// TIA Portal V15.1 export
// export: Created 2024-05-17T05:38:39.4621169Z, ExportSetting WithDefaults, DisplayName Totally Integrated Automation Portal, DisplayVersion V15.1 Update 5, DisplayName TIA Portal Openness, DisplayVersion V15.1 Update 5, DisplayName SINAMICS Startdrive Advanced, DisplayVersion V15.1, DisplayName G130, G150, S120, S150, SINAMICS MV, S210, DisplayVersion V15.1, DisplayName G110M, G120, G120C, G120D, G120P, DisplayVersion V15.1, DisplayName STEP 7 Professional, DisplayVersion V15.1 Update 5, DisplayName STEP 7 Safety, DisplayVersion V15.1, DisplayName WinCC Professional, DisplayVersion V15.1 Update 5, DisplayName SIMATIC Visualization Architect, DisplayVersion V15.1
FUNCTION_BLOCK "LGBBodyStopper"   // FB6666, FBD
TITLE = LGBBodyStopper
{ S7_Optimized_Access := 'FALSE' }
AUTHOR : Imtech
VERSION : 0.1
// stored: AutoNumber false, IsIECCheckEnabled false, SetENOAutomatically False, UDAEnableTagReadback false
   VAR_INPUT
      I_BodyNr { ExternalAccessible := 'False'; ExternalVisible := 'False'; ExternalWritable := 'False'} : DInt;   // Body Number
      I_ColorCodeBC { ExternalAccessible := 'False'; ExternalVisible := 'False'; ExternalWritable := 'False'} : DInt;   // Color BC
      I_ColorCodeCC { ExternalAccessible := 'False'; ExternalVisible := 'False'; ExternalWritable := 'False'} : DInt;   // Color CC
      I_MMFRUSS { ExternalAccessible := 'False'; ExternalVisible := 'False'; ExternalWritable := 'False'} : DInt;   // MMFRUSS
      I_StartSearch { ExternalAccessible := 'False'; ExternalVisible := 'False'; ExternalWritable := 'False'} : Bool;   // Start search function
      I_ClearSearch { ExternalAccessible := 'False'; ExternalVisible := 'False'; ExternalWritable := 'False'} : Bool;   // Clear search result
   END_VAR
   VAR_OUTPUT
      O_BodyGo { ExternalAccessible := 'False'; ExternalVisible := 'False'; ExternalWritable := 'False'} : Bool;   // Body can GO
      O_BodyStop { ExternalAccessible := 'False'; ExternalVisible := 'False'; ExternalWritable := 'False'} : Bool;   // Body must STOP
      O_AlarmABCondition { ExternalAccessible := 'False'; ExternalVisible := 'False'; ExternalWritable := 'False'} : Bool;   // Alarm AB condition
      O_AlarmA { ExternalAccessible := 'False'; ExternalVisible := 'False'; ExternalWritable := 'False'} : Bool;   // Alarms A
      O_AlarmB { ExternalAccessible := 'False'; ExternalVisible := 'False'; ExternalWritable := 'False'} : Bool;   // Alarms B
      O_AlarmC { ExternalAccessible := 'False'; ExternalVisible := 'False'; ExternalWritable := 'False'} : Bool;   // Alarms C
      O_AlarmD { ExternalAccessible := 'False'; ExternalVisible := 'False'; ExternalWritable := 'False'} : Bool;   // Alarms D
      H_AlarmDWord { ExternalAccessible := 'False'; ExternalVisible := 'False'; ExternalWritable := 'False'} : DWord;
   END_VAR
   VAR_IN_OUT
      H_HMI : "H_HMI";   // HMI Icon Animation
      H_GBBodyStopper : "H_GBBodyStopper";   // HMI Animation
   END_VAR
   VAR DB_SPECIFIC
      AC_BodyStop { ExternalAccessible := 'False'; ExternalVisible := 'False'; ExternalWritable := 'False'} : Bool;   // Body is stopped, there is a selection active
      BodyGo { ExternalAccessible := 'False'; ExternalVisible := 'False'; ExternalWritable := 'False'} : Bool;   // Body can Go
      BodyStop { ExternalAccessible := 'False'; ExternalVisible := 'False'; ExternalWritable := 'False'} : Bool;   // Body must Stop
      HMILayerGeneral { ExternalAccessible := 'False'; ExternalVisible := 'False'; ExternalWritable := 'False'} : Bool;
      HMILayerSealing { ExternalAccessible := 'False'; ExternalVisible := 'False'; ExternalWritable := 'False'} : Bool;
      HMILayerPaint { ExternalAccessible := 'False'; ExternalVisible := 'False'; ExternalWritable := 'False'} : Bool;
      HMICmdForce { ExternalAccessible := 'False'; ExternalVisible := 'False'; ExternalWritable := 'False'} : Bool;
      HMICmdJustR { ExternalAccessible := 'False'; ExternalVisible := 'False'; ExternalWritable := 'False'} : Bool;
      HMICmdJustS2 { ExternalAccessible := 'False'; ExternalVisible := 'False'; ExternalWritable := 'False'} : Bool;
      HMICmdMM1stLayer { ExternalAccessible := 'False'; ExternalVisible := 'False'; ExternalWritable := 'False'} : Bool;
      HMICmdMM2ndLayer { ExternalAccessible := 'False'; ExternalVisible := 'False'; ExternalWritable := 'False'} : Bool;
      Status_HMICmdForce { ExternalAccessible := 'False'; ExternalVisible := 'False'; ExternalWritable := 'False'} : Bool;
      Status_HMICmdMM1stLayer { ExternalAccessible := 'False'; ExternalVisible := 'False'; ExternalWritable := 'False'} : Bool;
      Status_HMICmdMM2ndLayer { ExternalAccessible := 'False'; ExternalVisible := 'False'; ExternalWritable := 'False'} : Bool;
      Status_TABGeneral { ExternalAccessible := 'False'; ExternalVisible := 'False'; ExternalWritable := 'False'} : Bool;
      Status_TABSealing { ExternalAccessible := 'False'; ExternalVisible := 'False'; ExternalWritable := 'False'} : Bool;
      Status_TABPaint { ExternalAccessible := 'False'; ExternalVisible := 'False'; ExternalWritable := 'False'} : Bool;
      MM { ExternalAccessible := 'False'; ExternalVisible := 'False'; ExternalWritable := 'False'} : Int;
      FR { ExternalAccessible := 'False'; ExternalVisible := 'False'; ExternalWritable := 'False'} : Int;
      USS { ExternalAccessible := 'False'; ExternalVisible := 'False'; ExternalWritable := 'False'} : Int;
      FRUSS { ExternalAccessible := 'False'; ExternalVisible := 'False'; ExternalWritable := 'False'} : DInt;
      M1 { ExternalAccessible := 'False'; ExternalVisible := 'False'; ExternalWritable := 'False'} : Int;
      M2 { ExternalAccessible := 'False'; ExternalVisible := 'False'; ExternalWritable := 'False'} : Int;
      F { ExternalAccessible := 'False'; ExternalVisible := 'False'; ExternalWritable := 'False'} : Int;
      R { ExternalAccessible := 'False'; ExternalVisible := 'False'; ExternalWritable := 'False'} : Int;
      U { ExternalAccessible := 'False'; ExternalVisible := 'False'; ExternalWritable := 'False'} : Int;
      S1 { ExternalAccessible := 'False'; ExternalVisible := 'False'; ExternalWritable := 'False'} : Int;
      S2 { ExternalAccessible := 'False'; ExternalVisible := 'False'; ExternalWritable := 'False'} : Int;
      Done { ExternalAccessible := 'False'; ExternalVisible := 'False'; ExternalWritable := 'False'} : Bool;
      Error { ExternalAccessible := 'False'; ExternalVisible := 'False'; ExternalWritable := 'False'} : Bool;
      ColorCodeBCShort { ExternalAccessible := 'False'; ExternalVisible := 'False'; ExternalWritable := 'False'} : DInt;   // Color BC
      NoDuoTone { ExternalAccessible := 'False'; ExternalVisible := 'False'; ExternalWritable := 'False'} : Bool;
      DuoTone1stLayer { ExternalAccessible := 'False'; ExternalVisible := 'False'; ExternalWritable := 'False'} : Bool;
      DuoTone2ndLayer { ExternalAccessible := 'False'; ExternalVisible := 'False'; ExternalWritable := 'False'} : Bool;
      InitBit { ExternalAccessible := 'False'; ExternalVisible := 'False'; ExternalWritable := 'False'} : Bool;
      AlarmABCondition { ExternalAccessible := 'False'; ExternalVisible := 'False'; ExternalWritable := 'False'} : Bool;
      AlarmA { ExternalAccessible := 'False'; ExternalVisible := 'False'; ExternalWritable := 'False'} : Bool;
      AlarmB { ExternalAccessible := 'False'; ExternalVisible := 'False'; ExternalWritable := 'False'} : Bool;
      AlarmC { ExternalAccessible := 'False'; ExternalVisible := 'False'; ExternalWritable := 'False'} : Bool;
      AlarmD { ExternalAccessible := 'False'; ExternalVisible := 'False'; ExternalWritable := 'False'} : Bool;
      ArrayHMI_BodyNr { ExternalAccessible := 'False'; ExternalVisible := 'False'; ExternalWritable := 'False'} : Array[1..10] of DInt;
      ArrayHMI_ColorCodeBC { ExternalAccessible := 'False'; ExternalVisible := 'False'; ExternalWritable := 'False'} : Array[1..10] of Int;
      ArrayHMI_ColorCodeCC { ExternalAccessible := 'False'; ExternalVisible := 'False'; ExternalWritable := 'False'} : Array[1..10] of Int;
      ArrayHMI_MM { ExternalAccessible := 'False'; ExternalVisible := 'False'; ExternalWritable := 'False'} : Array[1..10] of Int;
      ArrayHMI_MMwithR { ExternalAccessible := 'False'; ExternalVisible := 'False'; ExternalWritable := 'False'} : Array[1..10] of Int;
      ArrayHMI_MMwithS2 { ExternalAccessible := 'False'; ExternalVisible := 'False'; ExternalWritable := 'False'} : Array[1..10] of Int;
      ArrayHMI_R { ExternalAccessible := 'False'; ExternalVisible := 'False'; ExternalWritable := 'False'} : Array[1..10] of Int;
      ArrayHMI_S2 { ExternalAccessible := 'False'; ExternalVisible := 'False'; ExternalWritable := 'False'} : Array[1..10] of Int;
      ArrayHMI_DuoTone { ExternalAccessible := 'False'; ExternalVisible := 'False'; ExternalWritable := 'False'} : Array[1..10] of Int;
      Status_BodyNr { ExternalAccessible := 'False'; ExternalVisible := 'False'; ExternalWritable := 'False'} : Array[1..10] of Bool;
      Status_ColorCodeBC { ExternalAccessible := 'False'; ExternalVisible := 'False'; ExternalWritable := 'False'} : Array[1..10] of Bool;
      Status_ColorCodeCC { ExternalAccessible := 'False'; ExternalVisible := 'False'; ExternalWritable := 'False'} : Array[1..10] of Bool;
      Status_MM { ExternalAccessible := 'False'; ExternalVisible := 'False'; ExternalWritable := 'False'} : Array[1..10] of Bool;
      Status_MMwithR { ExternalAccessible := 'False'; ExternalVisible := 'False'; ExternalWritable := 'False'} : Array[1..10] of Bool;
      Status_MMwithS2 { ExternalAccessible := 'False'; ExternalVisible := 'False'; ExternalWritable := 'False'} : Array[1..10] of Bool;
   END_VAR
   VAR
      BodyStopperSub { ExternalAccessible := 'False'; ExternalVisible := 'False'; ExternalWritable := 'False'} : "LGBBodyStopperSub";   // LBodyStopperSub
   END_VAR
   VAR_TEMP   // added for the SCL form of the ladder/FBD networks
      _w1 : Bool;
      _w2 : Bool;
   END_VAR
BEGIN

REGION Network 1: **** 1 - Inputs **** Layer INIT
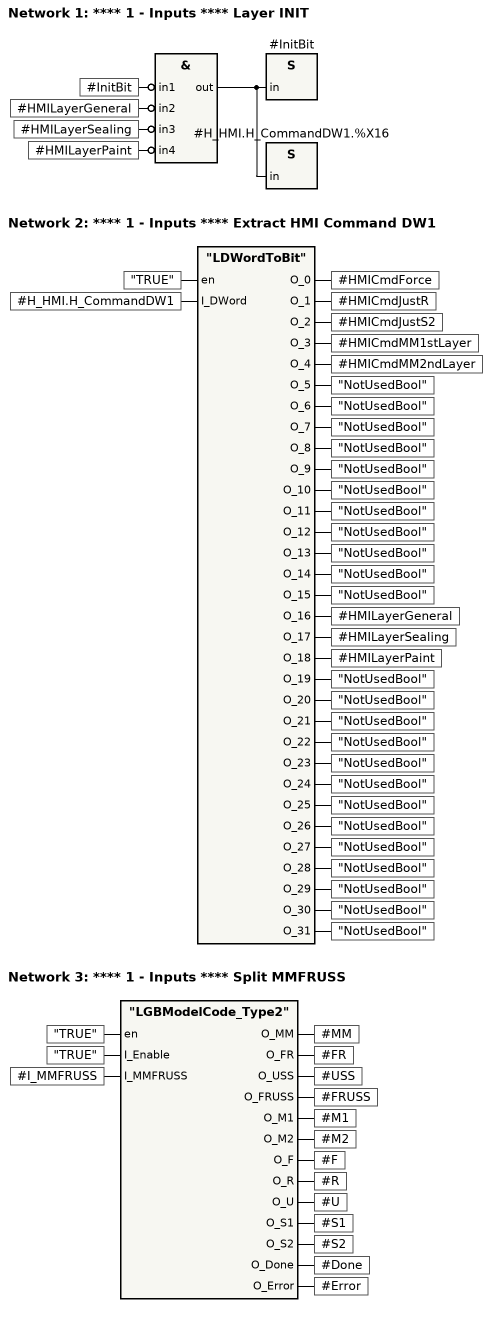
   #_w1 := NOT #InitBit AND NOT #HMILayerGeneral AND NOT #HMILayerSealing AND NOT #HMILayerPaint;
   IF #_w1 THEN
       #InitBit := TRUE;
       #H_HMI.H_CommandDW1.%X16 := TRUE;
   END_IF;
END_REGION

REGION Network 2: **** 1 - Inputs **** Extract HMI Command DW1
   IF "TRUE" THEN
       "LDWordToBit"(I_DWord := #H_HMI.H_CommandDW1,
                     O_0 => #HMICmdForce,
                     O_1 => #HMICmdJustR,
                     O_2 => #HMICmdJustS2,
                     O_3 => #HMICmdMM1stLayer,
                     O_4 => #HMICmdMM2ndLayer,
                     O_5 => "NotUsedBool",
                     O_6 => "NotUsedBool",
                     O_7 => "NotUsedBool",
                     O_8 => "NotUsedBool",
                     O_9 => "NotUsedBool",
                     O_10 => "NotUsedBool",
                     O_11 => "NotUsedBool",
                     O_12 => "NotUsedBool",
                     O_13 => "NotUsedBool",
                     O_14 => "NotUsedBool",
                     O_15 => "NotUsedBool",
                     O_16 => #HMILayerGeneral,
                     O_17 => #HMILayerSealing,
                     O_18 => #HMILayerPaint,
                     O_19 => "NotUsedBool",
                     O_20 => "NotUsedBool",
                     O_21 => "NotUsedBool",
                     O_22 => "NotUsedBool",
                     O_23 => "NotUsedBool",
                     O_24 => "NotUsedBool",
                     O_25 => "NotUsedBool",
                     O_26 => "NotUsedBool",
                     O_27 => "NotUsedBool",
                     O_28 => "NotUsedBool",
                     O_29 => "NotUsedBool",
                     O_30 => "NotUsedBool",
                     O_31 => "NotUsedBool");
   END_IF;
END_REGION

REGION Network 3: **** 1 - Inputs **** Split MMFRUSS
   IF "TRUE" THEN
       "LGBModelCode_Type2"(I_Enable := "TRUE",
                            I_MMFRUSS := #I_MMFRUSS,
                            O_MM => #MM,
                            O_FR => #FR,
                            O_USS => #USS,
                            O_FRUSS => #FRUSS,
                            O_M1 => #M1,
                            O_M2 => #M2,
                            O_F => #F,
                            O_R => #R,
                            O_U => #U,
                            O_S1 => #S1,
                            O_S2 => #S2,
                            O_Done => #Done,
                            O_Error => #Error);
   END_IF;
END_REGION

REGION Network 4: **** 1 - Inputs **** ColorCode BC Short
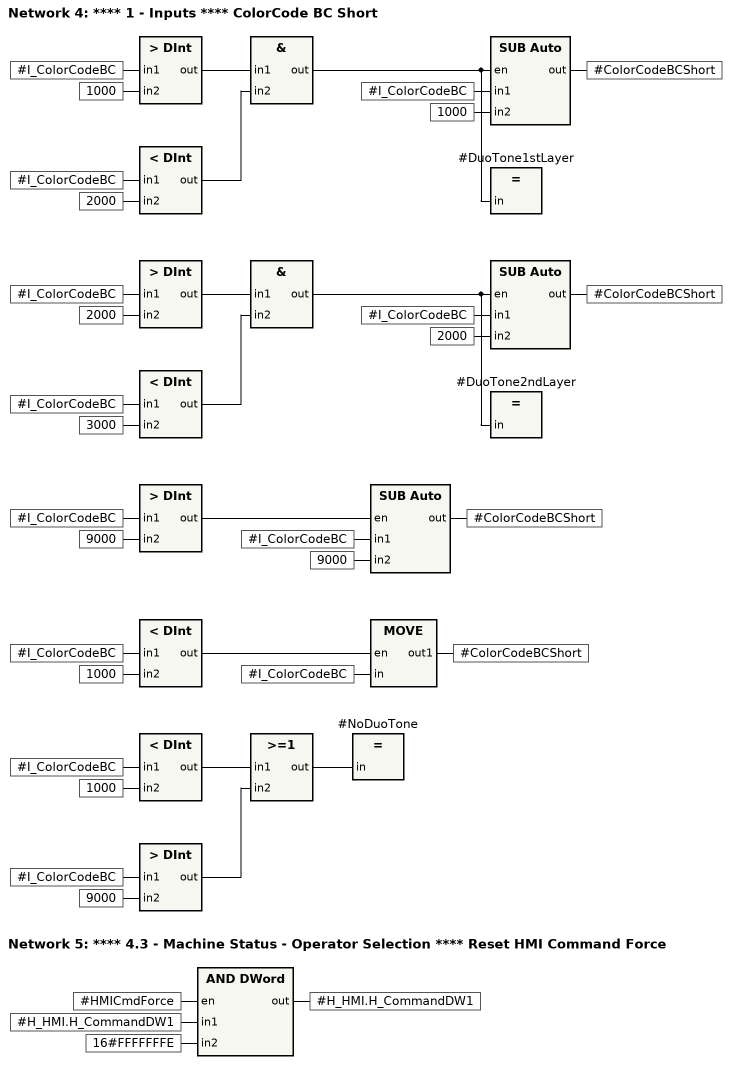
   #_w1 := (#I_ColorCodeBC > 1000) AND (#I_ColorCodeBC < 2000);
   IF #_w1 THEN #ColorCodeBCShort := #I_ColorCodeBC - 1000; END_IF;
   #DuoTone1stLayer := #_w1;
   #_w2 := (#I_ColorCodeBC > 2000) AND (#I_ColorCodeBC < 3000);
   IF #_w2 THEN #ColorCodeBCShort := #I_ColorCodeBC - 2000; END_IF;
   #DuoTone2ndLayer := #_w2;
   IF #I_ColorCodeBC > 9000 THEN #ColorCodeBCShort := #I_ColorCodeBC - 9000; END_IF;
   IF #I_ColorCodeBC < 1000 THEN #ColorCodeBCShort := #I_ColorCodeBC; END_IF;
   #NoDuoTone := (#I_ColorCodeBC < 1000) OR (#I_ColorCodeBC > 9000);
END_REGION

REGION Network 5: **** 4.3 - Machine Status - Operator Selection **** Reset HMI Command Force
   IF #HMICmdForce THEN #H_HMI.H_CommandDW1 := #H_HMI.H_CommandDW1 AND 16#FFFFFFFE; END_IF;
END_REGION

REGION Network 6: **** 4.6 - Machine status - Indications **** Animation DW1 General
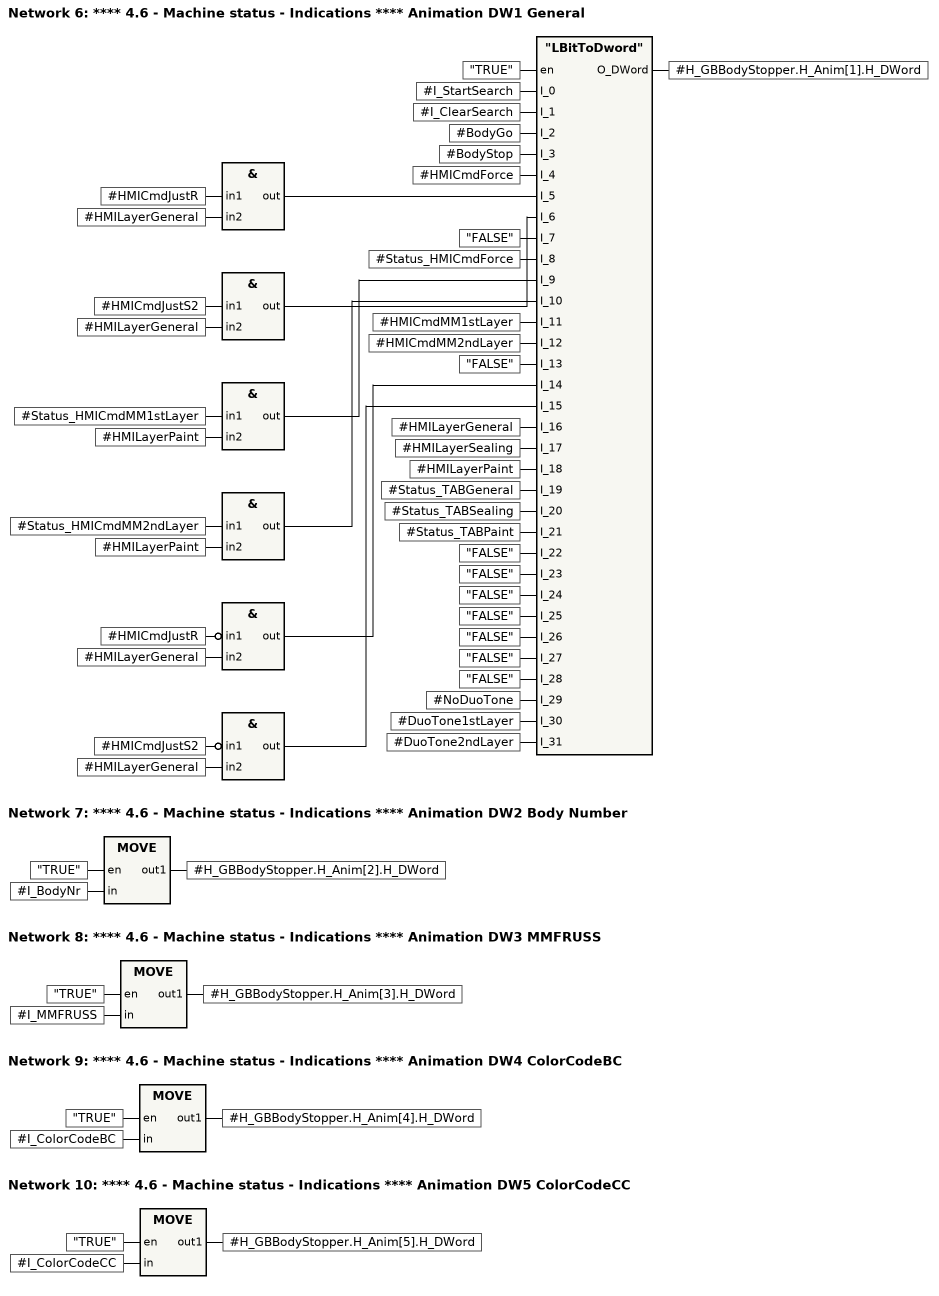
   IF "TRUE" THEN
       "LBitToDword"(I_0 := #I_StartSearch,
                     I_1 := #I_ClearSearch,
                     I_2 := #BodyGo,
                     I_3 := #BodyStop,
                     I_4 := #HMICmdForce,
                     I_5 := #HMICmdJustR AND #HMILayerGeneral,
                     I_6 := #HMICmdJustS2 AND #HMILayerGeneral,
                     I_7 := "FALSE",
                     I_8 := #Status_HMICmdForce,
                     I_9 := #Status_HMICmdMM1stLayer AND #HMILayerPaint,
                     I_10 := #Status_HMICmdMM2ndLayer AND #HMILayerPaint,
                     I_11 := #HMICmdMM1stLayer,
                     I_12 := #HMICmdMM2ndLayer,
                     I_13 := "FALSE",
                     I_14 := NOT #HMICmdJustR AND #HMILayerGeneral,
                     I_15 := NOT #HMICmdJustS2 AND #HMILayerGeneral,
                     I_16 := #HMILayerGeneral,
                     I_17 := #HMILayerSealing,
                     I_18 := #HMILayerPaint,
                     I_19 := #Status_TABGeneral,
                     I_20 := #Status_TABSealing,
                     I_21 := #Status_TABPaint,
                     I_22 := "FALSE",
                     I_23 := "FALSE",
                     I_24 := "FALSE",
                     I_25 := "FALSE",
                     I_26 := "FALSE",
                     I_27 := "FALSE",
                     I_28 := "FALSE",
                     I_29 := #NoDuoTone,
                     I_30 := #DuoTone1stLayer,
                     I_31 := #DuoTone2ndLayer,
                     O_DWord => #H_GBBodyStopper.H_Anim[1].H_DWord);
   END_IF;
END_REGION

REGION Network 7: **** 4.6 - Machine status - Indications **** Animation DW2 Body Number
   IF "TRUE" THEN #H_GBBodyStopper.H_Anim[2].H_DWord := #I_BodyNr; END_IF;
END_REGION

REGION Network 8: **** 4.6 - Machine status - Indications **** Animation DW3 MMFRUSS
   IF "TRUE" THEN #H_GBBodyStopper.H_Anim[3].H_DWord := #I_MMFRUSS; END_IF;
END_REGION

REGION Network 9: **** 4.6 - Machine status - Indications **** Animation DW4 ColorCodeBC
   IF "TRUE" THEN #H_GBBodyStopper.H_Anim[4].H_DWord := #I_ColorCodeBC; END_IF;
END_REGION

REGION Network 10: **** 4.6 - Machine status - Indications **** Animation DW5 ColorCodeCC
   IF "TRUE" THEN #H_GBBodyStopper.H_Anim[5].H_DWord := #I_ColorCodeCC; END_IF;
END_REGION

REGION Network 11: **** 4.6 - Machine status - Indications **** Animation DW6 ColorCodeBC Short
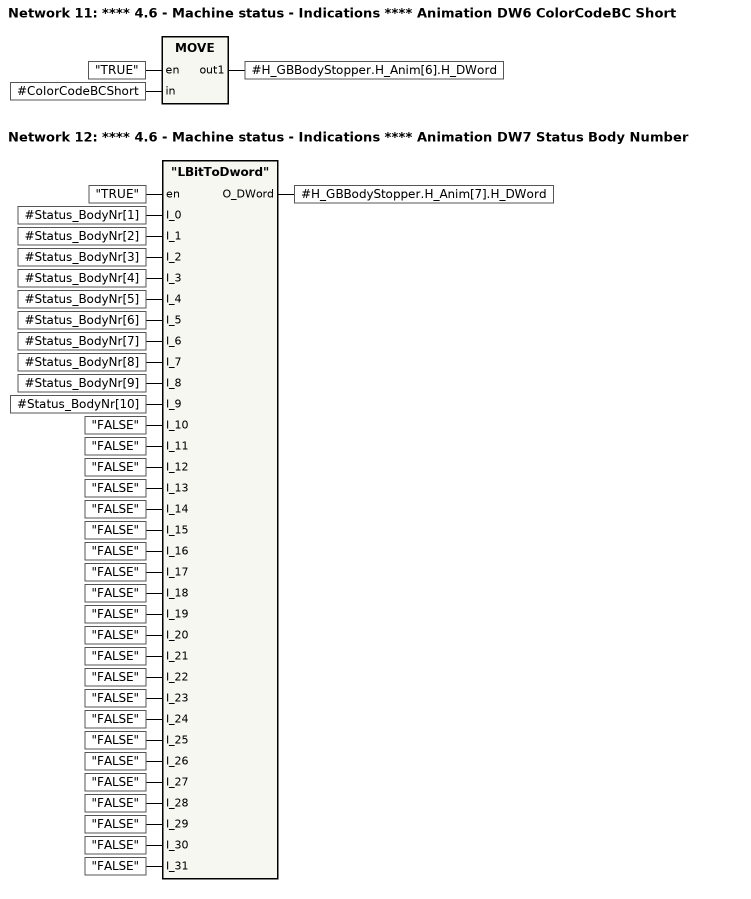
   IF "TRUE" THEN #H_GBBodyStopper.H_Anim[6].H_DWord := #ColorCodeBCShort; END_IF;
END_REGION

REGION Network 12: **** 4.6 - Machine status - Indications **** Animation DW7 Status Body Number
   IF "TRUE" THEN
       "LBitToDword"(I_0 := #Status_BodyNr[1],
                     I_1 := #Status_BodyNr[2],
                     I_2 := #Status_BodyNr[3],
                     I_3 := #Status_BodyNr[4],
                     I_4 := #Status_BodyNr[5],
                     I_5 := #Status_BodyNr[6],
                     I_6 := #Status_BodyNr[7],
                     I_7 := #Status_BodyNr[8],
                     I_8 := #Status_BodyNr[9],
                     I_9 := #Status_BodyNr[10],
                     I_10 := "FALSE",
                     I_11 := "FALSE",
                     I_12 := "FALSE",
                     I_13 := "FALSE",
                     I_14 := "FALSE",
                     I_15 := "FALSE",
                     I_16 := "FALSE",
                     I_17 := "FALSE",
                     I_18 := "FALSE",
                     I_19 := "FALSE",
                     I_20 := "FALSE",
                     I_21 := "FALSE",
                     I_22 := "FALSE",
                     I_23 := "FALSE",
                     I_24 := "FALSE",
                     I_25 := "FALSE",
                     I_26 := "FALSE",
                     I_27 := "FALSE",
                     I_28 := "FALSE",
                     I_29 := "FALSE",
                     I_30 := "FALSE",
                     I_31 := "FALSE",
                     O_DWord => #H_GBBodyStopper.H_Anim[7].H_DWord);
   END_IF;
END_REGION

REGION Network 13: **** 4.6 - Machine status - Indications **** Animation DW8 Status ColorCodeBC
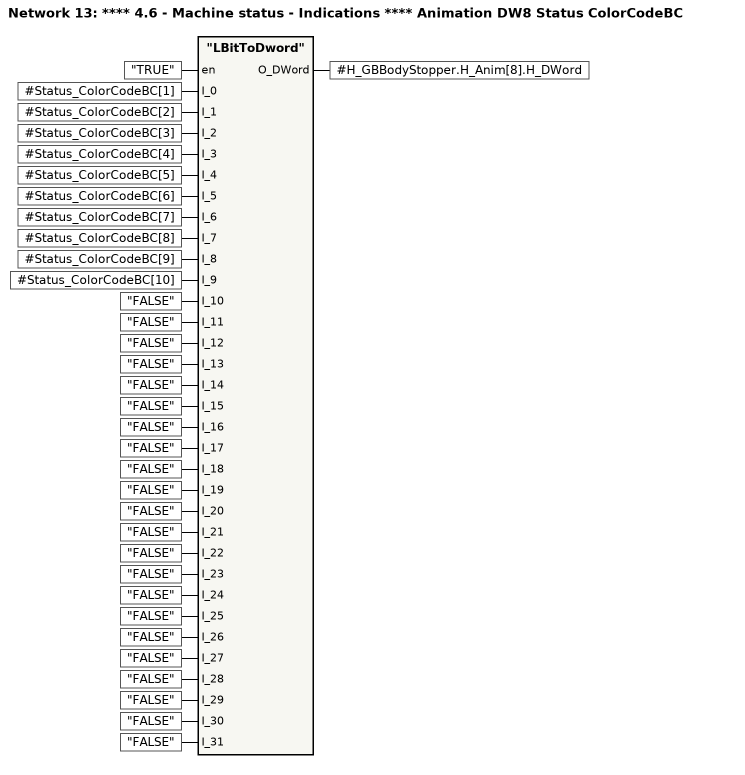
   IF "TRUE" THEN
       "LBitToDword"(I_0 := #Status_ColorCodeBC[1],
                     I_1 := #Status_ColorCodeBC[2],
                     I_2 := #Status_ColorCodeBC[3],
                     I_3 := #Status_ColorCodeBC[4],
                     I_4 := #Status_ColorCodeBC[5],
                     I_5 := #Status_ColorCodeBC[6],
                     I_6 := #Status_ColorCodeBC[7],
                     I_7 := #Status_ColorCodeBC[8],
                     I_8 := #Status_ColorCodeBC[9],
                     I_9 := #Status_ColorCodeBC[10],
                     I_10 := "FALSE",
                     I_11 := "FALSE",
                     I_12 := "FALSE",
                     I_13 := "FALSE",
                     I_14 := "FALSE",
                     I_15 := "FALSE",
                     I_16 := "FALSE",
                     I_17 := "FALSE",
                     I_18 := "FALSE",
                     I_19 := "FALSE",
                     I_20 := "FALSE",
                     I_21 := "FALSE",
                     I_22 := "FALSE",
                     I_23 := "FALSE",
                     I_24 := "FALSE",
                     I_25 := "FALSE",
                     I_26 := "FALSE",
                     I_27 := "FALSE",
                     I_28 := "FALSE",
                     I_29 := "FALSE",
                     I_30 := "FALSE",
                     I_31 := "FALSE",
                     O_DWord => #H_GBBodyStopper.H_Anim[8].H_DWord);
   END_IF;
END_REGION

REGION Network 14: **** 4.6 - Machine status - Indications **** Animation DW9 Status ColorCodeCC
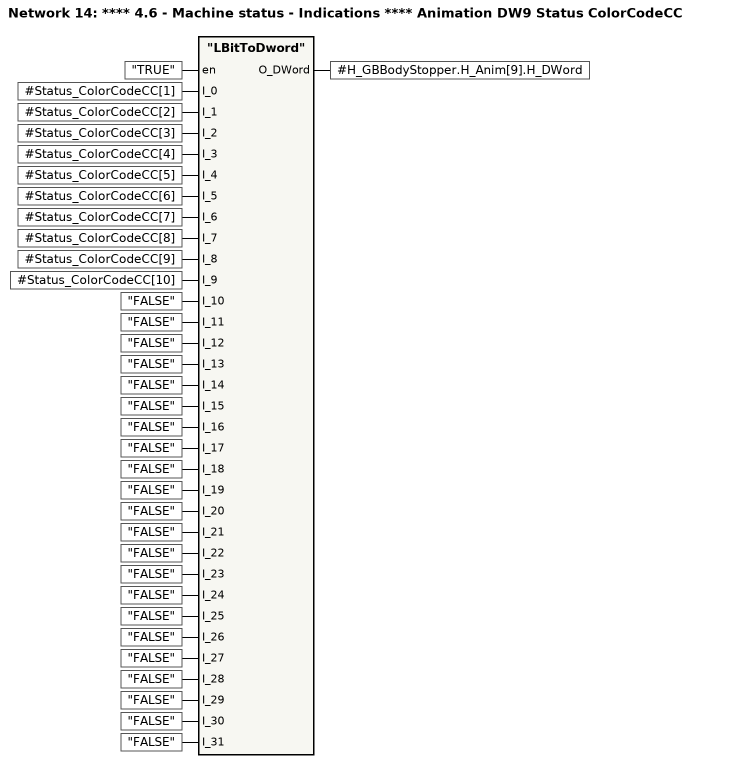
   IF "TRUE" THEN
       "LBitToDword"(I_0 := #Status_ColorCodeCC[1],
                     I_1 := #Status_ColorCodeCC[2],
                     I_2 := #Status_ColorCodeCC[3],
                     I_3 := #Status_ColorCodeCC[4],
                     I_4 := #Status_ColorCodeCC[5],
                     I_5 := #Status_ColorCodeCC[6],
                     I_6 := #Status_ColorCodeCC[7],
                     I_7 := #Status_ColorCodeCC[8],
                     I_8 := #Status_ColorCodeCC[9],
                     I_9 := #Status_ColorCodeCC[10],
                     I_10 := "FALSE",
                     I_11 := "FALSE",
                     I_12 := "FALSE",
                     I_13 := "FALSE",
                     I_14 := "FALSE",
                     I_15 := "FALSE",
                     I_16 := "FALSE",
                     I_17 := "FALSE",
                     I_18 := "FALSE",
                     I_19 := "FALSE",
                     I_20 := "FALSE",
                     I_21 := "FALSE",
                     I_22 := "FALSE",
                     I_23 := "FALSE",
                     I_24 := "FALSE",
                     I_25 := "FALSE",
                     I_26 := "FALSE",
                     I_27 := "FALSE",
                     I_28 := "FALSE",
                     I_29 := "FALSE",
                     I_30 := "FALSE",
                     I_31 := "FALSE",
                     O_DWord => #H_GBBodyStopper.H_Anim[9].H_DWord);
   END_IF;
END_REGION

REGION Network 15: **** 4.6 - Machine status - Indications **** Animation DW10 Status MM
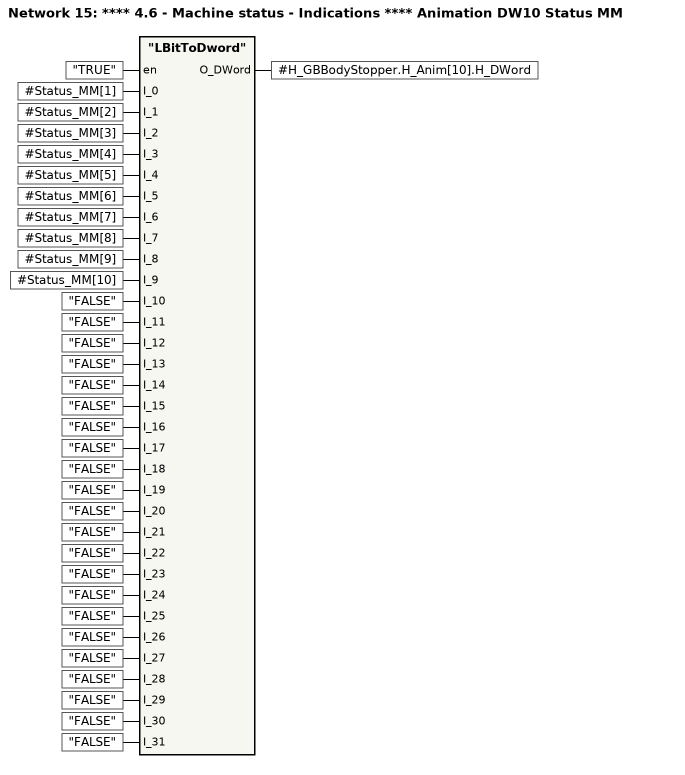
   IF "TRUE" THEN
       "LBitToDword"(I_0 := #Status_MM[1],
                     I_1 := #Status_MM[2],
                     I_2 := #Status_MM[3],
                     I_3 := #Status_MM[4],
                     I_4 := #Status_MM[5],
                     I_5 := #Status_MM[6],
                     I_6 := #Status_MM[7],
                     I_7 := #Status_MM[8],
                     I_8 := #Status_MM[9],
                     I_9 := #Status_MM[10],
                     I_10 := "FALSE",
                     I_11 := "FALSE",
                     I_12 := "FALSE",
                     I_13 := "FALSE",
                     I_14 := "FALSE",
                     I_15 := "FALSE",
                     I_16 := "FALSE",
                     I_17 := "FALSE",
                     I_18 := "FALSE",
                     I_19 := "FALSE",
                     I_20 := "FALSE",
                     I_21 := "FALSE",
                     I_22 := "FALSE",
                     I_23 := "FALSE",
                     I_24 := "FALSE",
                     I_25 := "FALSE",
                     I_26 := "FALSE",
                     I_27 := "FALSE",
                     I_28 := "FALSE",
                     I_29 := "FALSE",
                     I_30 := "FALSE",
                     I_31 := "FALSE",
                     O_DWord => #H_GBBodyStopper.H_Anim[10].H_DWord);
   END_IF;
END_REGION

REGION Network 16: **** 4.6 - Machine status - Indications **** Animation DW11 Status MM with R
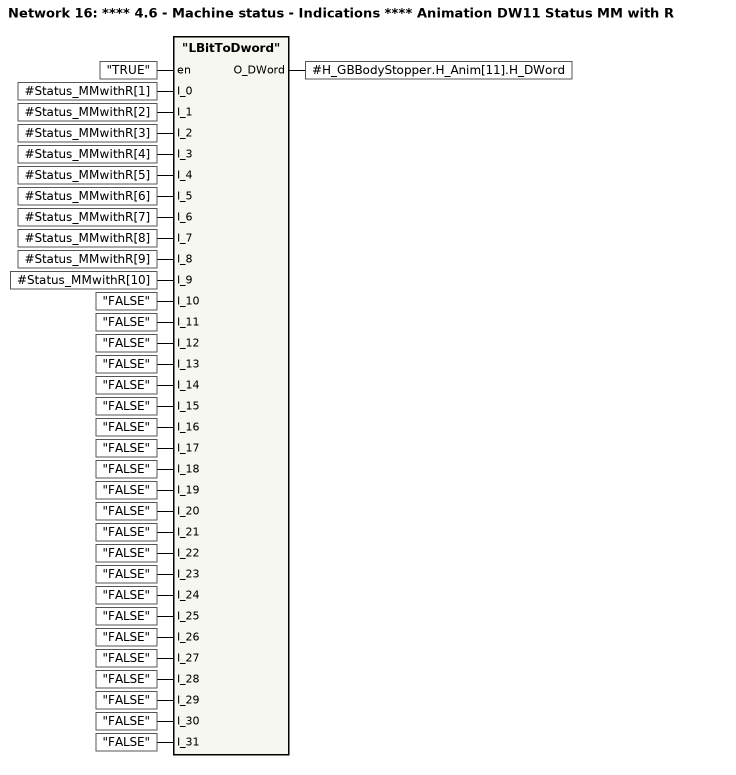
   IF "TRUE" THEN
       "LBitToDword"(I_0 := #Status_MMwithR[1],
                     I_1 := #Status_MMwithR[2],
                     I_2 := #Status_MMwithR[3],
                     I_3 := #Status_MMwithR[4],
                     I_4 := #Status_MMwithR[5],
                     I_5 := #Status_MMwithR[6],
                     I_6 := #Status_MMwithR[7],
                     I_7 := #Status_MMwithR[8],
                     I_8 := #Status_MMwithR[9],
                     I_9 := #Status_MMwithR[10],
                     I_10 := "FALSE",
                     I_11 := "FALSE",
                     I_12 := "FALSE",
                     I_13 := "FALSE",
                     I_14 := "FALSE",
                     I_15 := "FALSE",
                     I_16 := "FALSE",
                     I_17 := "FALSE",
                     I_18 := "FALSE",
                     I_19 := "FALSE",
                     I_20 := "FALSE",
                     I_21 := "FALSE",
                     I_22 := "FALSE",
                     I_23 := "FALSE",
                     I_24 := "FALSE",
                     I_25 := "FALSE",
                     I_26 := "FALSE",
                     I_27 := "FALSE",
                     I_28 := "FALSE",
                     I_29 := "FALSE",
                     I_30 := "FALSE",
                     I_31 := "FALSE",
                     O_DWord => #H_GBBodyStopper.H_Anim[11].H_DWord);
   END_IF;
END_REGION

REGION Network 17: **** 4.6 - Machine status - Indications **** Animation DW12 Status MM with S2
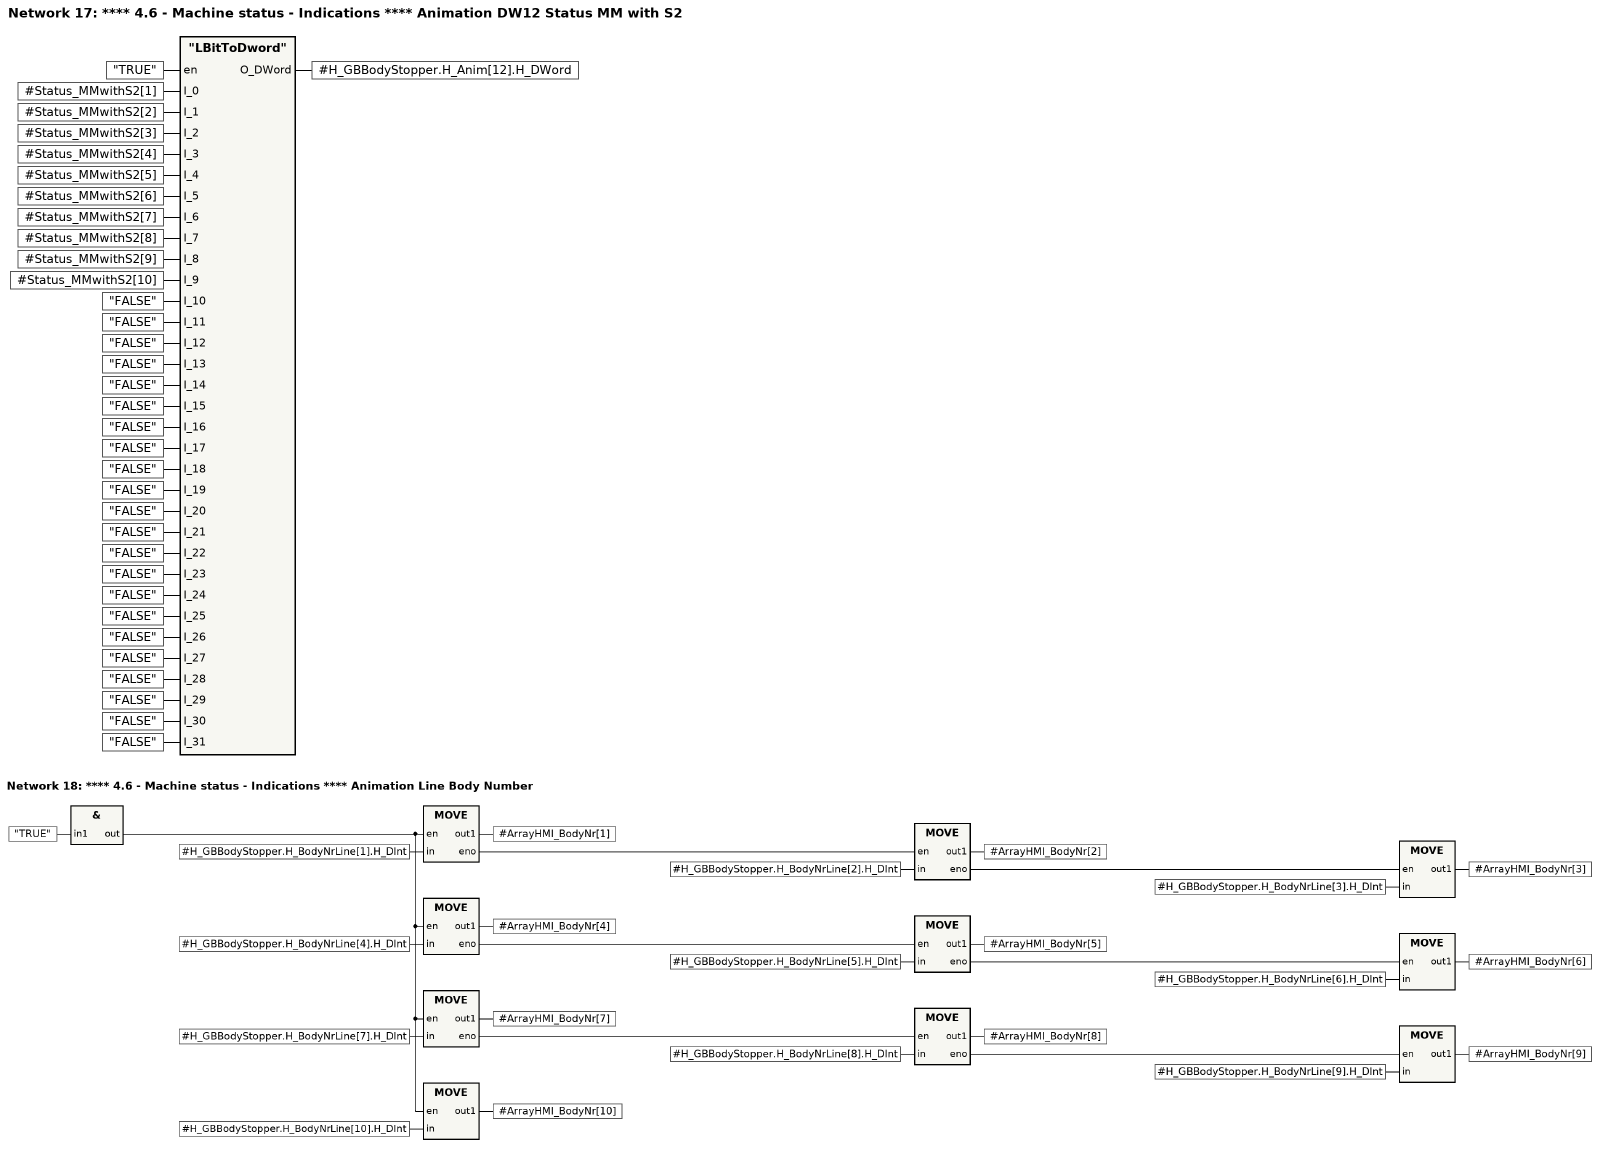
   IF "TRUE" THEN
       "LBitToDword"(I_0 := #Status_MMwithS2[1],
                     I_1 := #Status_MMwithS2[2],
                     I_2 := #Status_MMwithS2[3],
                     I_3 := #Status_MMwithS2[4],
                     I_4 := #Status_MMwithS2[5],
                     I_5 := #Status_MMwithS2[6],
                     I_6 := #Status_MMwithS2[7],
                     I_7 := #Status_MMwithS2[8],
                     I_8 := #Status_MMwithS2[9],
                     I_9 := #Status_MMwithS2[10],
                     I_10 := "FALSE",
                     I_11 := "FALSE",
                     I_12 := "FALSE",
                     I_13 := "FALSE",
                     I_14 := "FALSE",
                     I_15 := "FALSE",
                     I_16 := "FALSE",
                     I_17 := "FALSE",
                     I_18 := "FALSE",
                     I_19 := "FALSE",
                     I_20 := "FALSE",
                     I_21 := "FALSE",
                     I_22 := "FALSE",
                     I_23 := "FALSE",
                     I_24 := "FALSE",
                     I_25 := "FALSE",
                     I_26 := "FALSE",
                     I_27 := "FALSE",
                     I_28 := "FALSE",
                     I_29 := "FALSE",
                     I_30 := "FALSE",
                     I_31 := "FALSE",
                     O_DWord => #H_GBBodyStopper.H_Anim[12].H_DWord);
   END_IF;
END_REGION

REGION Network 18: **** 4.6 - Machine status - Indications **** Animation Line Body Number
   // ENO of a box is taken as its EN; it also drops when the box reports an error
   IF "TRUE" THEN
       #ArrayHMI_BodyNr[1] := #H_GBBodyStopper.H_BodyNrLine[1].H_DInt;
       #ArrayHMI_BodyNr[2] := #H_GBBodyStopper.H_BodyNrLine[2].H_DInt;
       #ArrayHMI_BodyNr[3] := #H_GBBodyStopper.H_BodyNrLine[3].H_DInt;
       #ArrayHMI_BodyNr[4] := #H_GBBodyStopper.H_BodyNrLine[4].H_DInt;
       #ArrayHMI_BodyNr[5] := #H_GBBodyStopper.H_BodyNrLine[5].H_DInt;
       #ArrayHMI_BodyNr[6] := #H_GBBodyStopper.H_BodyNrLine[6].H_DInt;
       #ArrayHMI_BodyNr[7] := #H_GBBodyStopper.H_BodyNrLine[7].H_DInt;
       #ArrayHMI_BodyNr[8] := #H_GBBodyStopper.H_BodyNrLine[8].H_DInt;
       #ArrayHMI_BodyNr[9] := #H_GBBodyStopper.H_BodyNrLine[9].H_DInt;
       #ArrayHMI_BodyNr[10] := #H_GBBodyStopper.H_BodyNrLine[10].H_DInt;
   END_IF;
END_REGION

REGION Network 19: **** 4.6 - Machine status - Indications **** Animation Line ColorCode BC
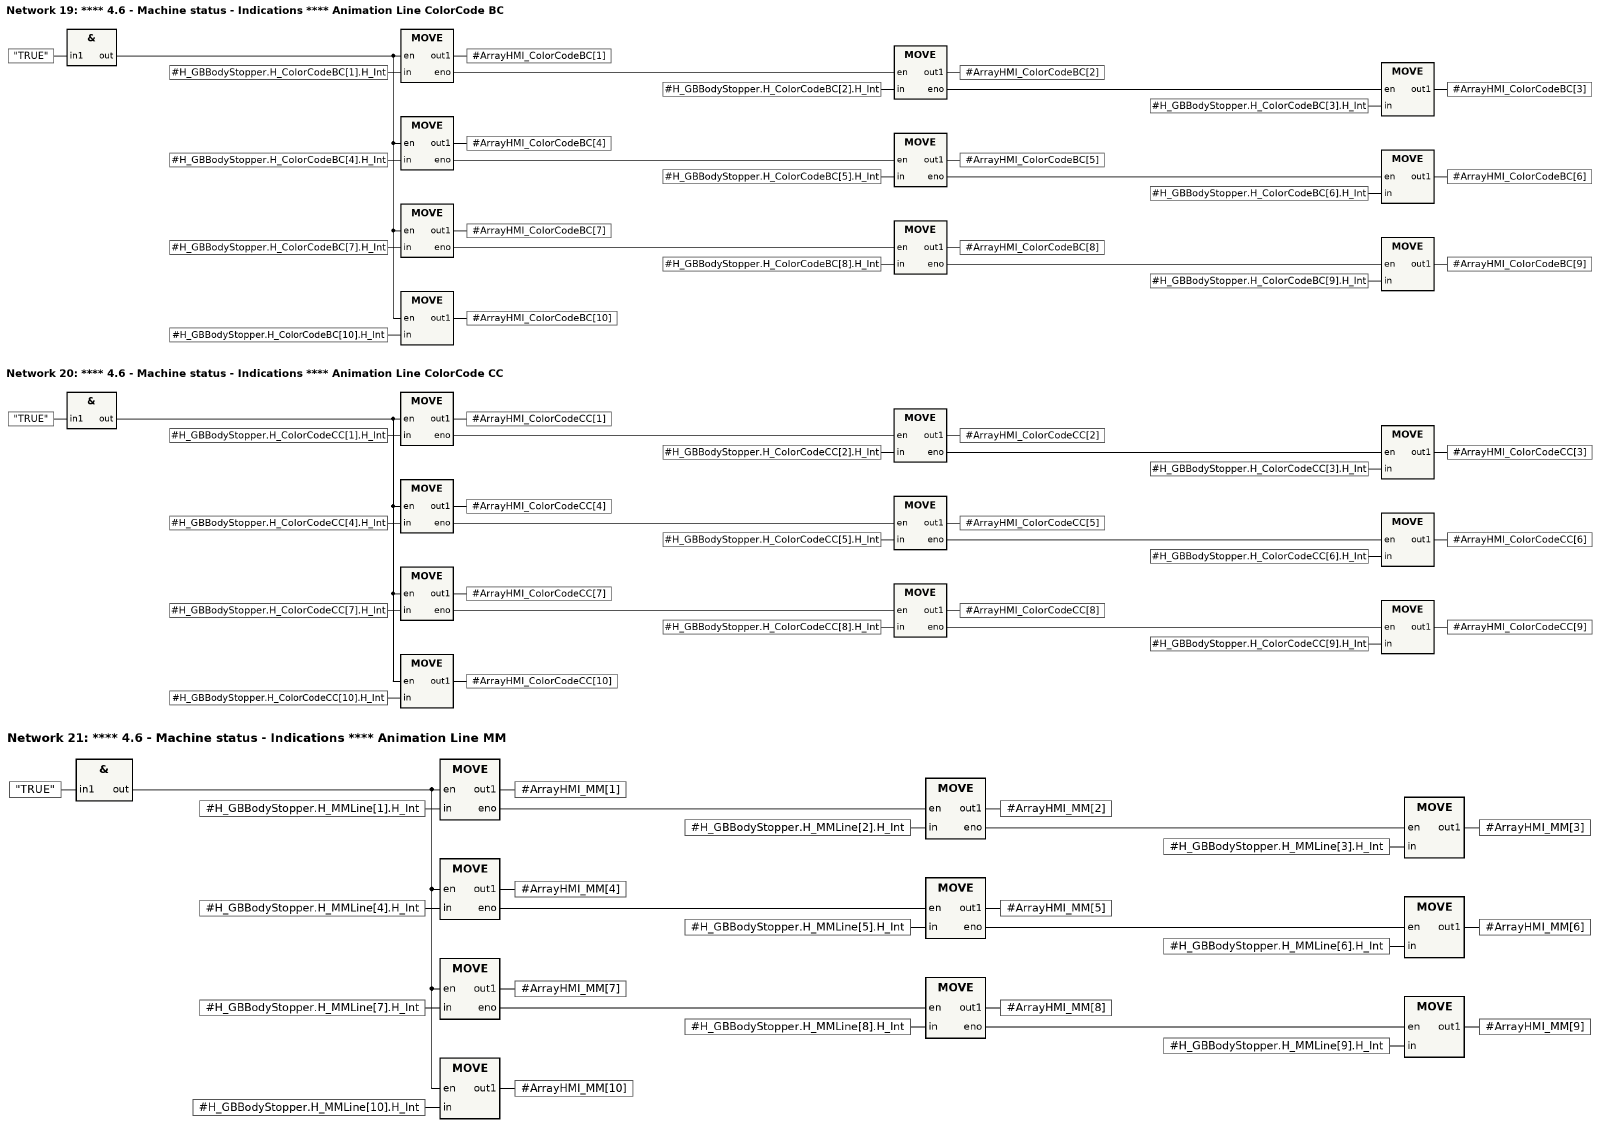
   // ENO of a box is taken as its EN; it also drops when the box reports an error
   IF "TRUE" THEN
       #ArrayHMI_ColorCodeBC[1] := #H_GBBodyStopper.H_ColorCodeBC[1].H_Int;
       #ArrayHMI_ColorCodeBC[2] := #H_GBBodyStopper.H_ColorCodeBC[2].H_Int;
       #ArrayHMI_ColorCodeBC[3] := #H_GBBodyStopper.H_ColorCodeBC[3].H_Int;
       #ArrayHMI_ColorCodeBC[4] := #H_GBBodyStopper.H_ColorCodeBC[4].H_Int;
       #ArrayHMI_ColorCodeBC[5] := #H_GBBodyStopper.H_ColorCodeBC[5].H_Int;
       #ArrayHMI_ColorCodeBC[6] := #H_GBBodyStopper.H_ColorCodeBC[6].H_Int;
       #ArrayHMI_ColorCodeBC[7] := #H_GBBodyStopper.H_ColorCodeBC[7].H_Int;
       #ArrayHMI_ColorCodeBC[8] := #H_GBBodyStopper.H_ColorCodeBC[8].H_Int;
       #ArrayHMI_ColorCodeBC[9] := #H_GBBodyStopper.H_ColorCodeBC[9].H_Int;
       #ArrayHMI_ColorCodeBC[10] := #H_GBBodyStopper.H_ColorCodeBC[10].H_Int;
   END_IF;
END_REGION

REGION Network 20: **** 4.6 - Machine status - Indications **** Animation Line ColorCode CC
   // ENO of a box is taken as its EN; it also drops when the box reports an error
   IF "TRUE" THEN
       #ArrayHMI_ColorCodeCC[1] := #H_GBBodyStopper.H_ColorCodeCC[1].H_Int;
       #ArrayHMI_ColorCodeCC[2] := #H_GBBodyStopper.H_ColorCodeCC[2].H_Int;
       #ArrayHMI_ColorCodeCC[3] := #H_GBBodyStopper.H_ColorCodeCC[3].H_Int;
       #ArrayHMI_ColorCodeCC[4] := #H_GBBodyStopper.H_ColorCodeCC[4].H_Int;
       #ArrayHMI_ColorCodeCC[5] := #H_GBBodyStopper.H_ColorCodeCC[5].H_Int;
       #ArrayHMI_ColorCodeCC[6] := #H_GBBodyStopper.H_ColorCodeCC[6].H_Int;
       #ArrayHMI_ColorCodeCC[7] := #H_GBBodyStopper.H_ColorCodeCC[7].H_Int;
       #ArrayHMI_ColorCodeCC[8] := #H_GBBodyStopper.H_ColorCodeCC[8].H_Int;
       #ArrayHMI_ColorCodeCC[9] := #H_GBBodyStopper.H_ColorCodeCC[9].H_Int;
       #ArrayHMI_ColorCodeCC[10] := #H_GBBodyStopper.H_ColorCodeCC[10].H_Int;
   END_IF;
END_REGION

REGION Network 21: **** 4.6 - Machine status - Indications **** Animation Line MM
   // ENO of a box is taken as its EN; it also drops when the box reports an error
   IF "TRUE" THEN
       #ArrayHMI_MM[1] := #H_GBBodyStopper.H_MMLine[1].H_Int;
       #ArrayHMI_MM[2] := #H_GBBodyStopper.H_MMLine[2].H_Int;
       #ArrayHMI_MM[3] := #H_GBBodyStopper.H_MMLine[3].H_Int;
       #ArrayHMI_MM[4] := #H_GBBodyStopper.H_MMLine[4].H_Int;
       #ArrayHMI_MM[5] := #H_GBBodyStopper.H_MMLine[5].H_Int;
       #ArrayHMI_MM[6] := #H_GBBodyStopper.H_MMLine[6].H_Int;
       #ArrayHMI_MM[7] := #H_GBBodyStopper.H_MMLine[7].H_Int;
       #ArrayHMI_MM[8] := #H_GBBodyStopper.H_MMLine[8].H_Int;
       #ArrayHMI_MM[9] := #H_GBBodyStopper.H_MMLine[9].H_Int;
       #ArrayHMI_MM[10] := #H_GBBodyStopper.H_MMLine[10].H_Int;
   END_IF;
END_REGION

REGION Network 22: **** 4.6 - Machine status - Indications **** Animation Line MM with R
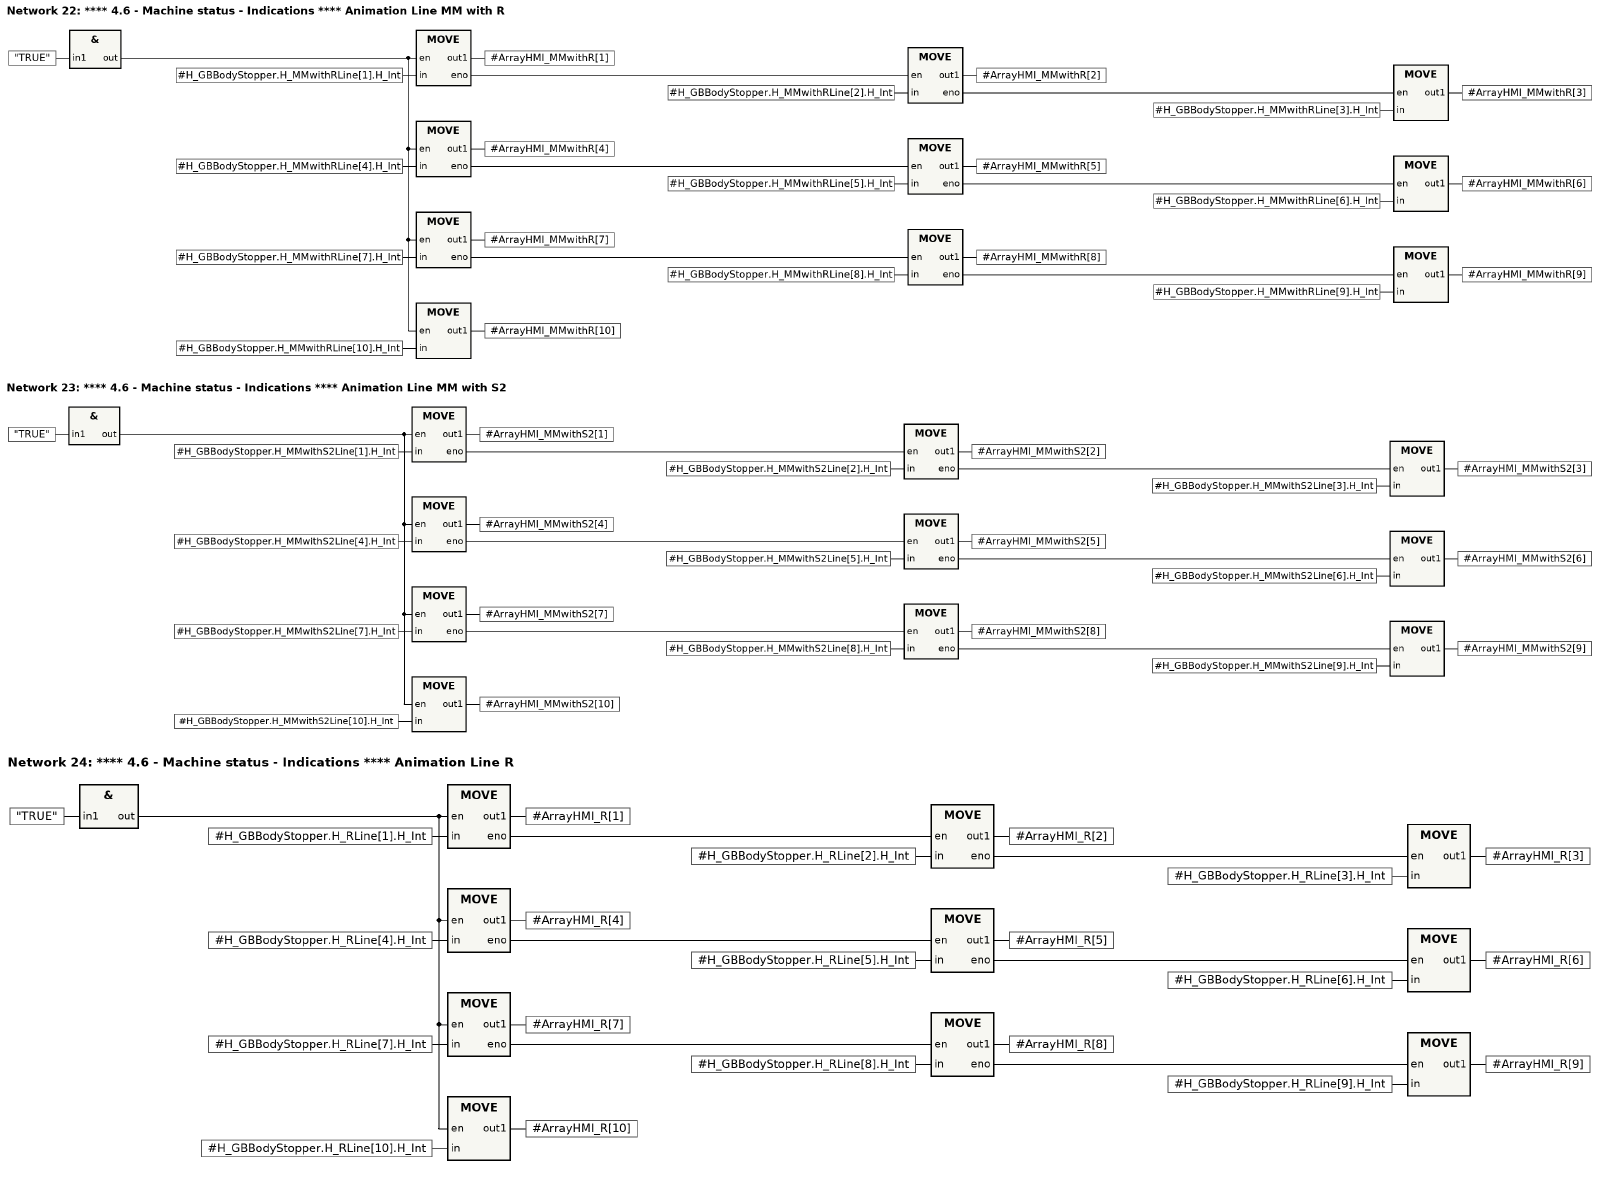
   // ENO of a box is taken as its EN; it also drops when the box reports an error
   IF "TRUE" THEN
       #ArrayHMI_MMwithR[1] := #H_GBBodyStopper.H_MMwithRLine[1].H_Int;
       #ArrayHMI_MMwithR[2] := #H_GBBodyStopper.H_MMwithRLine[2].H_Int;
       #ArrayHMI_MMwithR[3] := #H_GBBodyStopper.H_MMwithRLine[3].H_Int;
       #ArrayHMI_MMwithR[4] := #H_GBBodyStopper.H_MMwithRLine[4].H_Int;
       #ArrayHMI_MMwithR[5] := #H_GBBodyStopper.H_MMwithRLine[5].H_Int;
       #ArrayHMI_MMwithR[6] := #H_GBBodyStopper.H_MMwithRLine[6].H_Int;
       #ArrayHMI_MMwithR[7] := #H_GBBodyStopper.H_MMwithRLine[7].H_Int;
       #ArrayHMI_MMwithR[8] := #H_GBBodyStopper.H_MMwithRLine[8].H_Int;
       #ArrayHMI_MMwithR[9] := #H_GBBodyStopper.H_MMwithRLine[9].H_Int;
       #ArrayHMI_MMwithR[10] := #H_GBBodyStopper.H_MMwithRLine[10].H_Int;
   END_IF;
END_REGION

REGION Network 23: **** 4.6 - Machine status - Indications **** Animation Line MM with S2
   // ENO of a box is taken as its EN; it also drops when the box reports an error
   IF "TRUE" THEN
       #ArrayHMI_MMwithS2[1] := #H_GBBodyStopper.H_MMwithS2Line[1].H_Int;
       #ArrayHMI_MMwithS2[2] := #H_GBBodyStopper.H_MMwithS2Line[2].H_Int;
       #ArrayHMI_MMwithS2[3] := #H_GBBodyStopper.H_MMwithS2Line[3].H_Int;
       #ArrayHMI_MMwithS2[4] := #H_GBBodyStopper.H_MMwithS2Line[4].H_Int;
       #ArrayHMI_MMwithS2[5] := #H_GBBodyStopper.H_MMwithS2Line[5].H_Int;
       #ArrayHMI_MMwithS2[6] := #H_GBBodyStopper.H_MMwithS2Line[6].H_Int;
       #ArrayHMI_MMwithS2[7] := #H_GBBodyStopper.H_MMwithS2Line[7].H_Int;
       #ArrayHMI_MMwithS2[8] := #H_GBBodyStopper.H_MMwithS2Line[8].H_Int;
       #ArrayHMI_MMwithS2[9] := #H_GBBodyStopper.H_MMwithS2Line[9].H_Int;
       #ArrayHMI_MMwithS2[10] := #H_GBBodyStopper.H_MMwithS2Line[10].H_Int;
   END_IF;
END_REGION

REGION Network 24: **** 4.6 - Machine status - Indications **** Animation Line R
   // ENO of a box is taken as its EN; it also drops when the box reports an error
   IF "TRUE" THEN
       #ArrayHMI_R[1] := #H_GBBodyStopper.H_RLine[1].H_Int;
       #ArrayHMI_R[2] := #H_GBBodyStopper.H_RLine[2].H_Int;
       #ArrayHMI_R[3] := #H_GBBodyStopper.H_RLine[3].H_Int;
       #ArrayHMI_R[4] := #H_GBBodyStopper.H_RLine[4].H_Int;
       #ArrayHMI_R[5] := #H_GBBodyStopper.H_RLine[5].H_Int;
       #ArrayHMI_R[6] := #H_GBBodyStopper.H_RLine[6].H_Int;
       #ArrayHMI_R[7] := #H_GBBodyStopper.H_RLine[7].H_Int;
       #ArrayHMI_R[8] := #H_GBBodyStopper.H_RLine[8].H_Int;
       #ArrayHMI_R[9] := #H_GBBodyStopper.H_RLine[9].H_Int;
       #ArrayHMI_R[10] := #H_GBBodyStopper.H_RLine[10].H_Int;
   END_IF;
END_REGION

REGION Network 25: **** 4.6 - Machine status - Indications **** Animation Line S2
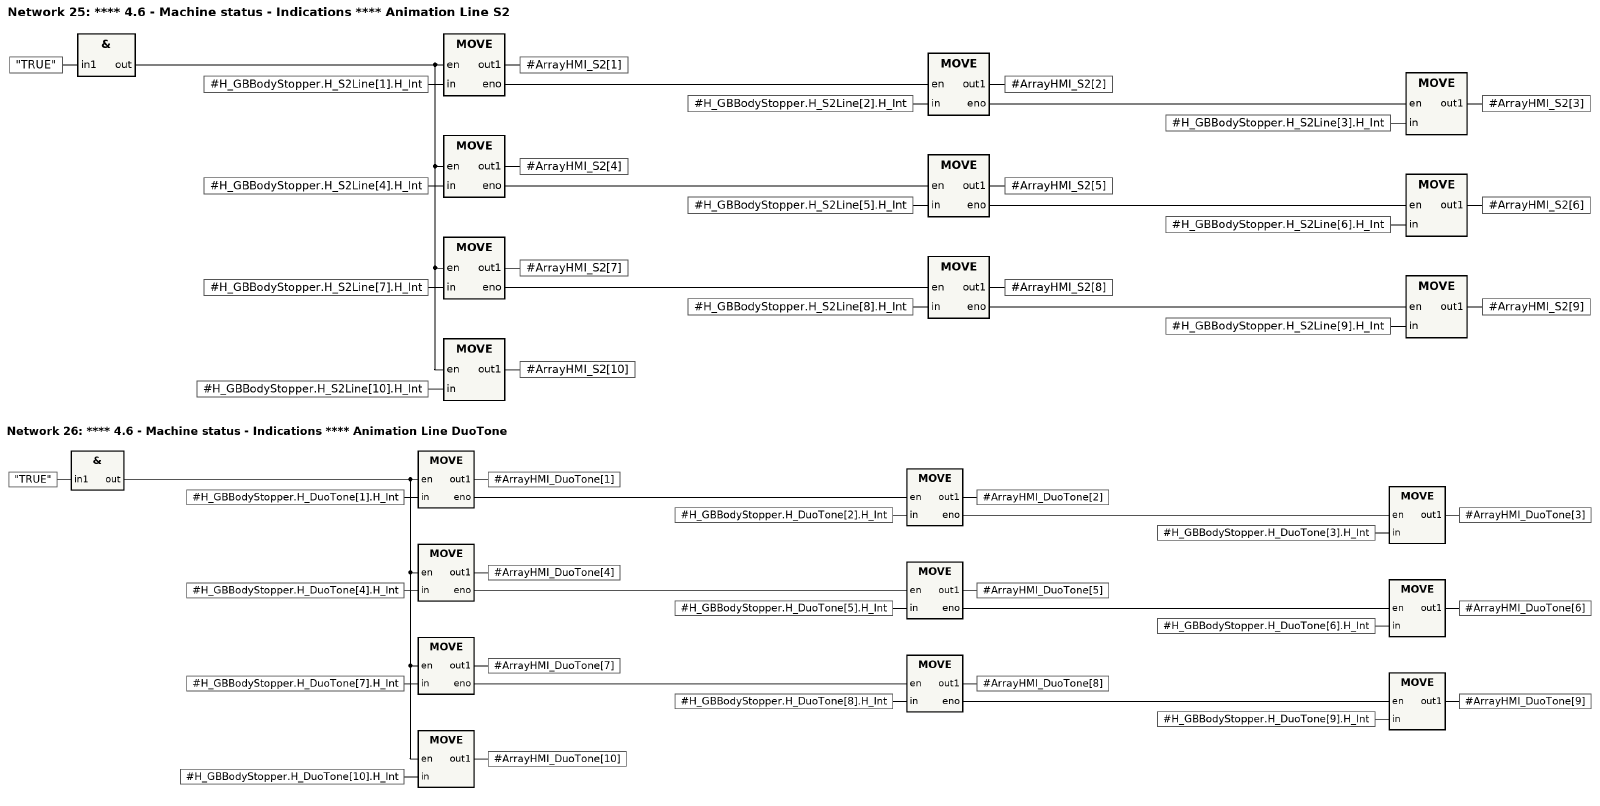
   // ENO of a box is taken as its EN; it also drops when the box reports an error
   IF "TRUE" THEN
       #ArrayHMI_S2[1] := #H_GBBodyStopper.H_S2Line[1].H_Int;
       #ArrayHMI_S2[2] := #H_GBBodyStopper.H_S2Line[2].H_Int;
       #ArrayHMI_S2[3] := #H_GBBodyStopper.H_S2Line[3].H_Int;
       #ArrayHMI_S2[4] := #H_GBBodyStopper.H_S2Line[4].H_Int;
       #ArrayHMI_S2[5] := #H_GBBodyStopper.H_S2Line[5].H_Int;
       #ArrayHMI_S2[6] := #H_GBBodyStopper.H_S2Line[6].H_Int;
       #ArrayHMI_S2[7] := #H_GBBodyStopper.H_S2Line[7].H_Int;
       #ArrayHMI_S2[8] := #H_GBBodyStopper.H_S2Line[8].H_Int;
       #ArrayHMI_S2[9] := #H_GBBodyStopper.H_S2Line[9].H_Int;
       #ArrayHMI_S2[10] := #H_GBBodyStopper.H_S2Line[10].H_Int;
   END_IF;
END_REGION

REGION Network 26: **** 4.6 - Machine status - Indications **** Animation Line DuoTone
   // ENO of a box is taken as its EN; it also drops when the box reports an error
   IF "TRUE" THEN
       #ArrayHMI_DuoTone[1] := #H_GBBodyStopper.H_DuoTone[1].H_Int;
       #ArrayHMI_DuoTone[2] := #H_GBBodyStopper.H_DuoTone[2].H_Int;
       #ArrayHMI_DuoTone[3] := #H_GBBodyStopper.H_DuoTone[3].H_Int;
       #ArrayHMI_DuoTone[4] := #H_GBBodyStopper.H_DuoTone[4].H_Int;
       #ArrayHMI_DuoTone[5] := #H_GBBodyStopper.H_DuoTone[5].H_Int;
       #ArrayHMI_DuoTone[6] := #H_GBBodyStopper.H_DuoTone[6].H_Int;
       #ArrayHMI_DuoTone[7] := #H_GBBodyStopper.H_DuoTone[7].H_Int;
       #ArrayHMI_DuoTone[8] := #H_GBBodyStopper.H_DuoTone[8].H_Int;
       #ArrayHMI_DuoTone[9] := #H_GBBodyStopper.H_DuoTone[9].H_Int;
       #ArrayHMI_DuoTone[10] := #H_GBBodyStopper.H_DuoTone[10].H_Int;
   END_IF;
END_REGION

REGION Network 27: **** 4.6 - Machine status - Indications **** Animation Line DuoTone
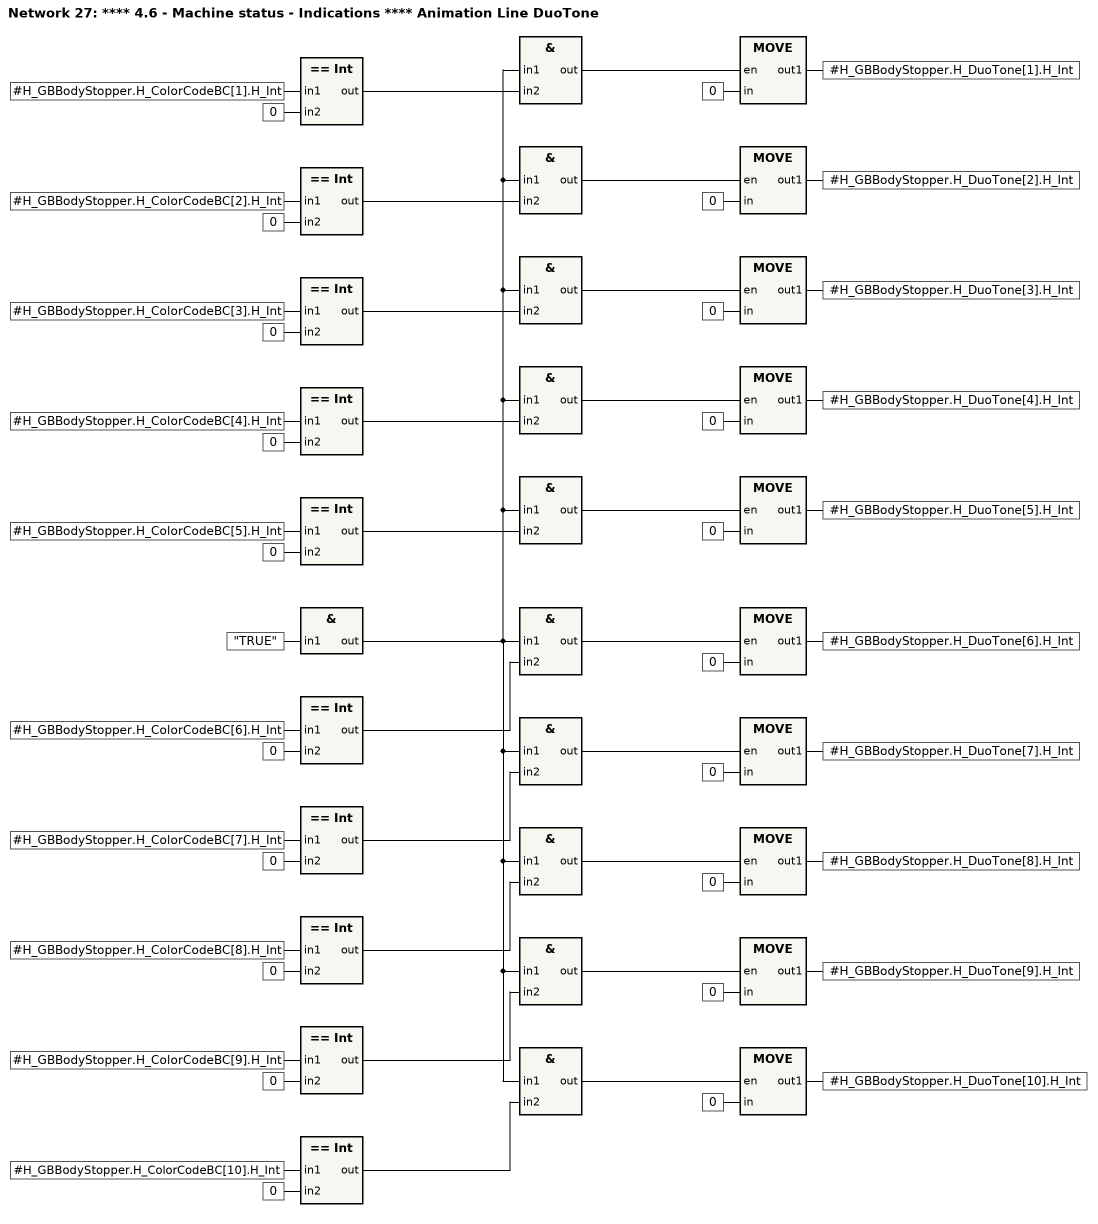
   IF "TRUE" AND (#H_GBBodyStopper.H_ColorCodeBC[1].H_Int = 0) THEN
       #H_GBBodyStopper.H_DuoTone[1].H_Int := 0;
   END_IF;
   IF "TRUE" AND (#H_GBBodyStopper.H_ColorCodeBC[2].H_Int = 0) THEN
       #H_GBBodyStopper.H_DuoTone[2].H_Int := 0;
   END_IF;
   IF "TRUE" AND (#H_GBBodyStopper.H_ColorCodeBC[3].H_Int = 0) THEN
       #H_GBBodyStopper.H_DuoTone[3].H_Int := 0;
   END_IF;
   IF "TRUE" AND (#H_GBBodyStopper.H_ColorCodeBC[4].H_Int = 0) THEN
       #H_GBBodyStopper.H_DuoTone[4].H_Int := 0;
   END_IF;
   IF "TRUE" AND (#H_GBBodyStopper.H_ColorCodeBC[5].H_Int = 0) THEN
       #H_GBBodyStopper.H_DuoTone[5].H_Int := 0;
   END_IF;
   IF "TRUE" AND (#H_GBBodyStopper.H_ColorCodeBC[6].H_Int = 0) THEN
       #H_GBBodyStopper.H_DuoTone[6].H_Int := 0;
   END_IF;
   IF "TRUE" AND (#H_GBBodyStopper.H_ColorCodeBC[7].H_Int = 0) THEN
       #H_GBBodyStopper.H_DuoTone[7].H_Int := 0;
   END_IF;
   IF "TRUE" AND (#H_GBBodyStopper.H_ColorCodeBC[8].H_Int = 0) THEN
       #H_GBBodyStopper.H_DuoTone[8].H_Int := 0;
   END_IF;
   IF "TRUE" AND (#H_GBBodyStopper.H_ColorCodeBC[9].H_Int = 0) THEN
       #H_GBBodyStopper.H_DuoTone[9].H_Int := 0;
   END_IF;
   IF "TRUE" AND (#H_GBBodyStopper.H_ColorCodeBC[10].H_Int = 0) THEN
       #H_GBBodyStopper.H_DuoTone[10].H_Int := 0;
   END_IF;
END_REGION

REGION Network 28: **** 4.6 - Machine status - Indications **** HMI Icon Animation
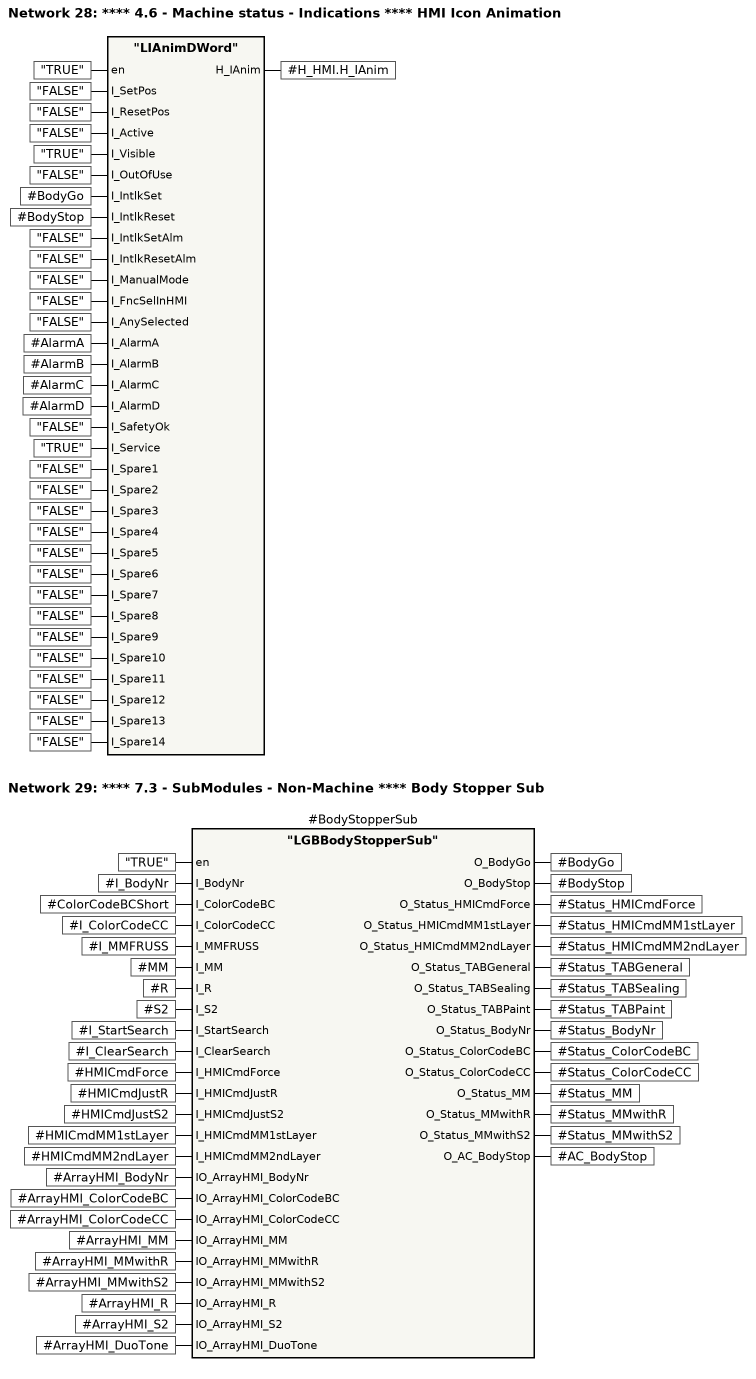
   IF "TRUE" THEN
       "LIAnimDWord"(I_SetPos := "FALSE",
                     I_ResetPos := "FALSE",
                     I_Active := "FALSE",
                     I_Visible := "TRUE",
                     I_OutOfUse := "FALSE",
                     I_IntlkSet := #BodyGo,
                     I_IntlkReset := #BodyStop,
                     I_IntlkSetAlm := "FALSE",
                     I_IntlkResetAlm := "FALSE",
                     I_ManualMode := "FALSE",
                     I_FncSelInHMI := "FALSE",
                     I_AnySelected := "FALSE",
                     I_AlarmA := #AlarmA,
                     I_AlarmB := #AlarmB,
                     I_AlarmC := #AlarmC,
                     I_AlarmD := #AlarmD,
                     I_SafetyOk := "FALSE",
                     I_Service := "TRUE",
                     I_Spare1 := "FALSE",
                     I_Spare2 := "FALSE",
                     I_Spare3 := "FALSE",
                     I_Spare4 := "FALSE",
                     I_Spare5 := "FALSE",
                     I_Spare6 := "FALSE",
                     I_Spare7 := "FALSE",
                     I_Spare8 := "FALSE",
                     I_Spare9 := "FALSE",
                     I_Spare10 := "FALSE",
                     I_Spare11 := "FALSE",
                     I_Spare12 := "FALSE",
                     I_Spare13 := "FALSE",
                     I_Spare14 := "FALSE",
                     H_IAnim => #H_HMI.H_IAnim);
   END_IF;
END_REGION

REGION Network 29: **** 7.3 - SubModules - Non-Machine **** Body Stopper Sub
   IF "TRUE" THEN
       #BodyStopperSub(I_BodyNr := #I_BodyNr,   // "LGBBodyStopperSub"
                       I_ColorCodeBC := #ColorCodeBCShort,
                       I_ColorCodeCC := #I_ColorCodeCC,
                       I_MMFRUSS := #I_MMFRUSS,
                       I_MM := #MM,
                       I_R := #R,
                       I_S2 := #S2,
                       I_StartSearch := #I_StartSearch,
                       I_ClearSearch := #I_ClearSearch,
                       I_HMICmdForce := #HMICmdForce,
                       I_HMICmdJustR := #HMICmdJustR,
                       I_HMICmdJustS2 := #HMICmdJustS2,
                       I_HMICmdMM1stLayer := #HMICmdMM1stLayer,
                       I_HMICmdMM2ndLayer := #HMICmdMM2ndLayer,
                       IO_ArrayHMI_BodyNr := #ArrayHMI_BodyNr,
                       IO_ArrayHMI_ColorCodeBC := #ArrayHMI_ColorCodeBC,
                       IO_ArrayHMI_ColorCodeCC := #ArrayHMI_ColorCodeCC,
                       IO_ArrayHMI_MM := #ArrayHMI_MM,
                       IO_ArrayHMI_MMwithR := #ArrayHMI_MMwithR,
                       IO_ArrayHMI_MMwithS2 := #ArrayHMI_MMwithS2,
                       IO_ArrayHMI_R := #ArrayHMI_R,
                       IO_ArrayHMI_S2 := #ArrayHMI_S2,
                       IO_ArrayHMI_DuoTone := #ArrayHMI_DuoTone,
                       O_BodyGo => #BodyGo,
                       O_BodyStop => #BodyStop,
                       O_Status_HMICmdForce => #Status_HMICmdForce,
                       O_Status_HMICmdMM1stLayer => #Status_HMICmdMM1stLayer,
                       O_Status_HMICmdMM2ndLayer => #Status_HMICmdMM2ndLayer,
                       O_Status_TABGeneral => #Status_TABGeneral,
                       O_Status_TABSealing => #Status_TABSealing,
                       O_Status_TABPaint => #Status_TABPaint,
                       O_Status_BodyNr => #Status_BodyNr,
                       O_Status_ColorCodeBC => #Status_ColorCodeBC,
                       O_Status_ColorCodeCC => #Status_ColorCodeCC,
                       O_Status_MM => #Status_MM,
                       O_Status_MMwithR => #Status_MMwithR,
                       O_Status_MMwithS2 => #Status_MMwithS2,
                       O_AC_BodyStop => #AC_BodyStop);
   END_IF;
END_REGION

REGION Network 30: **** 8 - Outputs **** Body Go
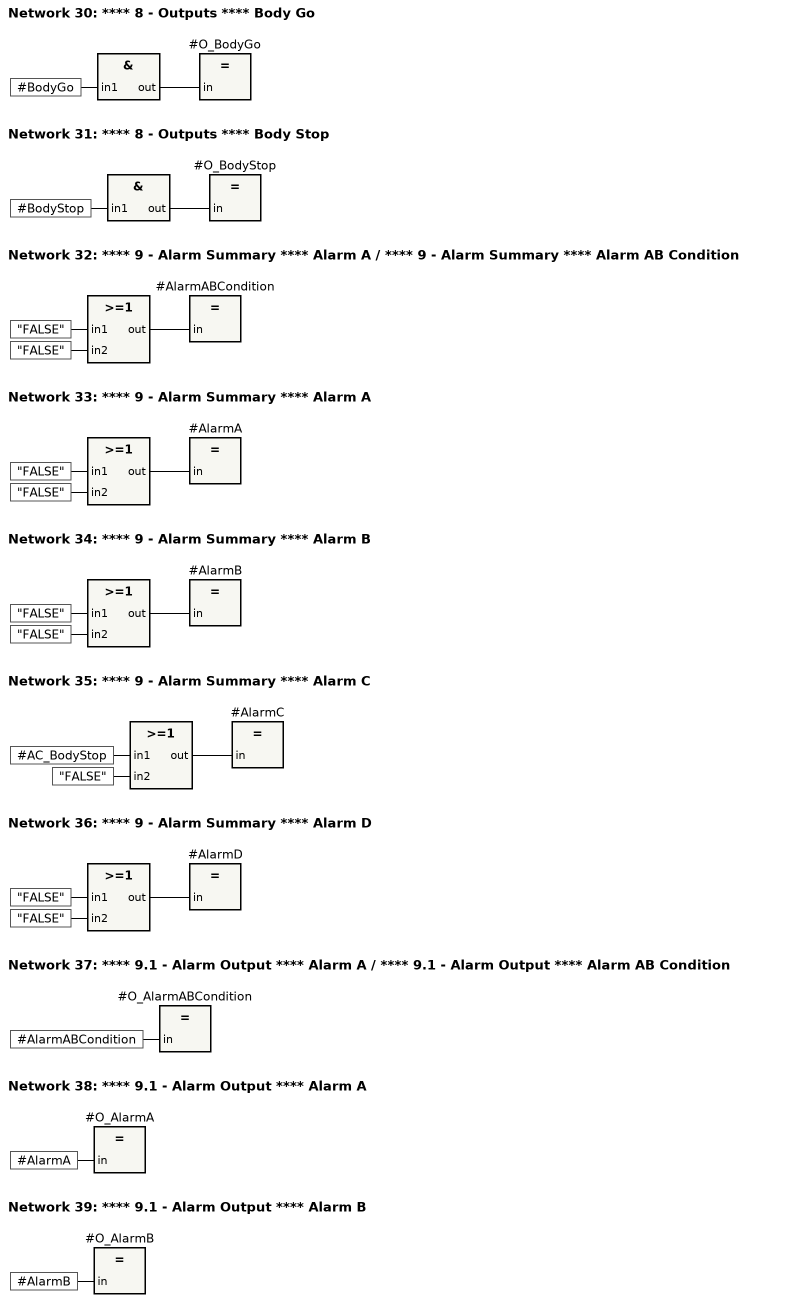
   #O_BodyGo := #BodyGo;
END_REGION

REGION Network 31: **** 8 - Outputs **** Body Stop
   #O_BodyStop := #BodyStop;
END_REGION

REGION Network 32: **** 9 - Alarm Summary **** Alarm A / **** 9 - Alarm Summary **** Alarm AB Condition
   // Alarm A
   #AlarmABCondition := "FALSE" OR "FALSE";
END_REGION

REGION Network 33: **** 9 - Alarm Summary **** Alarm A
   // Alarm A
   #AlarmA := "FALSE" OR "FALSE";
END_REGION

REGION Network 34: **** 9 - Alarm Summary **** Alarm B
   // Alarm B
   #AlarmB := "FALSE" OR "FALSE";
END_REGION

REGION Network 35: **** 9 - Alarm Summary **** Alarm C
   // Alarm C
   #AlarmC := #AC_BodyStop OR "FALSE";
END_REGION

REGION Network 36: **** 9 - Alarm Summary **** Alarm D
   // Alarm D
   #AlarmD := "FALSE" OR "FALSE";
END_REGION

REGION Network 37: **** 9.1 - Alarm Output **** Alarm A / **** 9.1 - Alarm Output **** Alarm AB Condition
   // Alarm A
   #O_AlarmABCondition := #AlarmABCondition;
END_REGION

REGION Network 38: **** 9.1 - Alarm Output **** Alarm A
   // Alarm A
   #O_AlarmA := #AlarmA;
END_REGION

REGION Network 39: **** 9.1 - Alarm Output **** Alarm B
   // Alarm B
   #O_AlarmB := #AlarmB;
END_REGION

REGION Network 40: **** 9.1 - Alarm Output **** Alarm C
   // Alarm C
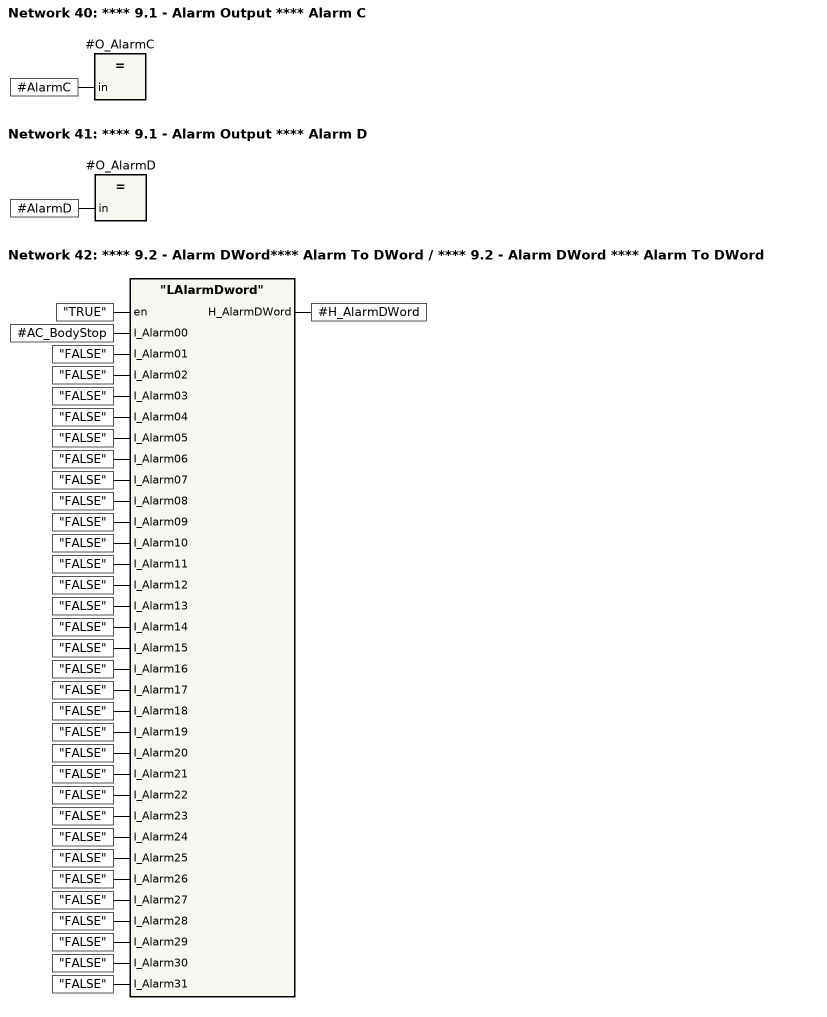
   #O_AlarmC := #AlarmC;
END_REGION

REGION Network 41: **** 9.1 - Alarm Output **** Alarm D
   // Alarm D
   #O_AlarmD := #AlarmD;
END_REGION

REGION Network 42: **** 9.2 - Alarm DWord**** Alarm To DWord / **** 9.2 - Alarm DWord **** Alarm To DWord
   // Alarm To Word
   IF "TRUE" THEN
       "LAlarmDword"(I_Alarm00 := #AC_BodyStop,
                     I_Alarm01 := "FALSE",
                     I_Alarm02 := "FALSE",
                     I_Alarm03 := "FALSE",
                     I_Alarm04 := "FALSE",
                     I_Alarm05 := "FALSE",
                     I_Alarm06 := "FALSE",
                     I_Alarm07 := "FALSE",
                     I_Alarm08 := "FALSE",
                     I_Alarm09 := "FALSE",
                     I_Alarm10 := "FALSE",
                     I_Alarm11 := "FALSE",
                     I_Alarm12 := "FALSE",
                     I_Alarm13 := "FALSE",
                     I_Alarm14 := "FALSE",
                     I_Alarm15 := "FALSE",
                     I_Alarm16 := "FALSE",
                     I_Alarm17 := "FALSE",
                     I_Alarm18 := "FALSE",
                     I_Alarm19 := "FALSE",
                     I_Alarm20 := "FALSE",
                     I_Alarm21 := "FALSE",
                     I_Alarm22 := "FALSE",
                     I_Alarm23 := "FALSE",
                     I_Alarm24 := "FALSE",
                     I_Alarm25 := "FALSE",
                     I_Alarm26 := "FALSE",
                     I_Alarm27 := "FALSE",
                     I_Alarm28 := "FALSE",
                     I_Alarm29 := "FALSE",
                     I_Alarm30 := "FALSE",
                     I_Alarm31 := "FALSE",
                     H_AlarmDWord => #H_AlarmDWord);
   END_IF;
END_REGION
END_FUNCTION_BLOCK
